{attribute 'GeneratedUsingTerminal: EPP2349-0021-0016'}
{attribute addProperty BoxType "EPP2349-0021-0016"}
{attribute addProperty Id "EtcSlaveTerminalBaseChannel_1AT %I*Channel_830843C11Channel_2AT %I*Channel_830843C11Channel_3AT %I*Channel_830843C11Channel_4AT %I*Channel_830843C11Channel_5AT %I*Channel_830843C11Channel_6AT %I*Channel_830843C11Channel_7AT %I*Channel_830843C11Channel_8AT %I*Channel_830843C11Channel_9AT %I*Channel_830843C11Channel_10AT %I*Channel_830843C11Channel_11AT %I*Channel_830843C11Channel_12AT %I*Channel_830843C11Channel_13AT %I*Channel_830843C11Channel_14AT %I*Channel_830843C11Channel_15AT %I*Channel_830843C11Channel_16AT %I*Channel_830843C11Channel_9_1AT %Q*Channel_42CA91F71Channel_10_1AT %Q*Channel_42CA91F71Channel_11_1AT %Q*Channel_42CA91F71Channel_12_1AT %Q*Channel_42CA91F71Channel_13_1AT %Q*Channel_42CA91F71Channel_14_1AT %Q*Channel_42CA91F71Channel_15_1AT %Q*Channel_42CA91F71Channel_16_1AT %Q*Channel_42CA91F71Channel_25AT %Q*Channel_42CA91F71Channel_26AT %Q*Channel_42CA91F71Channel_27AT %Q*Channel_42CA91F71Channel_28AT %Q*Channel_42CA91F71Channel_29AT %Q*Channel_42CA91F71Channel_30AT %Q*Channel_42CA91F71Channel_31AT %Q*Channel_42CA91F71Channel_32AT %Q*Channel_42CA91F71WcStateAT %I*WcState_9091E0EB2InfoDataAT %I*InfoData_6F19DB2B2"}
{attribute addProperty CRC "1636741124"}
{attribute addProperty Size "36"}
TYPE EPP2349_618EB004 EXTENDS EtcSlaveTerminalBase :
STRUCT
	{attribute addProperty Name "Channel_1"}
	Channel_1 : Channel_830843C1;
	{attribute addProperty Name "Channel_2"}
	Channel_2 : Channel_830843C1;
	{attribute addProperty Name "Channel_3"}
	Channel_3 : Channel_830843C1;
	{attribute addProperty Name "Channel_4"}
	Channel_4 : Channel_830843C1;
	{attribute addProperty Name "Channel_5"}
	Channel_5 : Channel_830843C1;
	{attribute addProperty Name "Channel_6"}
	Channel_6 : Channel_830843C1;
	{attribute addProperty Name "Channel_7"}
	Channel_7 : Channel_830843C1;
	{attribute addProperty Name "Channel_8"}
	Channel_8 : Channel_830843C1;
	{attribute addProperty Name "Channel_9"}
	Channel_9 : Channel_830843C1;
	{attribute addProperty Name "Channel_10"}
	Channel_10 : Channel_830843C1;
	{attribute addProperty Name "Channel_11"}
	Channel_11 : Channel_830843C1;
	{attribute addProperty Name "Channel_12"}
	Channel_12 : Channel_830843C1;
	{attribute addProperty Name "Channel_13"}
	Channel_13 : Channel_830843C1;
	{attribute addProperty Name "Channel_14"}
	Channel_14 : Channel_830843C1;
	{attribute addProperty Name "Channel_15"}
	Channel_15 : Channel_830843C1;
	{attribute addProperty Name "Channel_16"}
	Channel_16 : Channel_830843C1;
	{attribute addProperty Name "Channel_9_1"}
	Channel_9_1 : Channel_42CA91F7;
	{attribute addProperty Name "Channel_10_1"}
	Channel_10_1 : Channel_42CA91F7;
	{attribute addProperty Name "Channel_11_1"}
	Channel_11_1 : Channel_42CA91F7;
	{attribute addProperty Name "Channel_12_1"}
	Channel_12_1 : Channel_42CA91F7;
	{attribute addProperty Name "Channel_13_1"}
	Channel_13_1 : Channel_42CA91F7;
	{attribute addProperty Name "Channel_14_1"}
	Channel_14_1 : Channel_42CA91F7;
	{attribute addProperty Name "Channel_15_1"}
	Channel_15_1 : Channel_42CA91F7;
	{attribute addProperty Name "Channel_16_1"}
	Channel_16_1 : Channel_42CA91F7;
	{attribute addProperty Name "Channel_25"}
	Channel_25 : Channel_42CA91F7;
	{attribute addProperty Name "Channel_26"}
	Channel_26 : Channel_42CA91F7;
	{attribute addProperty Name "Channel_27"}
	Channel_27 : Channel_42CA91F7;
	{attribute addProperty Name "Channel_28"}
	Channel_28 : Channel_42CA91F7;
	{attribute addProperty Name "Channel_29"}
	Channel_29 : Channel_42CA91F7;
	{attribute addProperty Name "Channel_30"}
	Channel_30 : Channel_42CA91F7;
	{attribute addProperty Name "Channel_31"}
	Channel_31 : Channel_42CA91F7;
	{attribute addProperty Name "Channel_32"}
	Channel_32 : Channel_42CA91F7;
	{attribute addProperty Name "WcState"}
	WcState : WcState_9091E0EB;
	{attribute addProperty Name "InfoData"}
	InfoData : InfoData_6F19DB2B;
END_STRUCT
END_TYPE

(* stored: Version 1.2.0.0, ProductVersion 3.1.4024.9
   DUT EPP2349_618EB004: Id {09d2123e-a638-4db6-b49c-bef914296129} *)
